{attribute 'qualified_only'}
TYPE ePSBhardware :
(
	Wago := 0,
	Beckhoff := 1
); 
END_TYPE

(* stored: Version 1.1.0.1, ProductVersion 3.1.4024.12
   DUT ePSBhardware: Id {1ffebeca-da12-42cc-a254-8a9c7d82d500} *)
